// TIA Portal V17 export
// export: Created 2021-12-03T08:12:53.967625Z, ExportSetting WithDefaults, DisplayName Totally Integrated Automation Portal, DisplayVersion V17, DisplayName TIA Portal Openness, DisplayVersion V17, DisplayName TIA Portal Version Control Interface, DisplayVersion V17, DisplayName STEP 7 Professional, DisplayVersion V17, DisplayName STEP 7 Safety, DisplayVersion V17, DisplayName WinCC Advanced, DisplayVersion V17
FUNCTION "FC_DetLineCommunication_V2" : Void   // FC20, FBD
VERSION : 0.1
// stored: AutoNumber false, IsIECCheckEnabled false, UDAEnableTagReadback false
   VAR CONSTANT
      Speed_Convert : Int := 6;
   END_VAR
BEGIN

REGION Network 1: Detector Line: Start Request
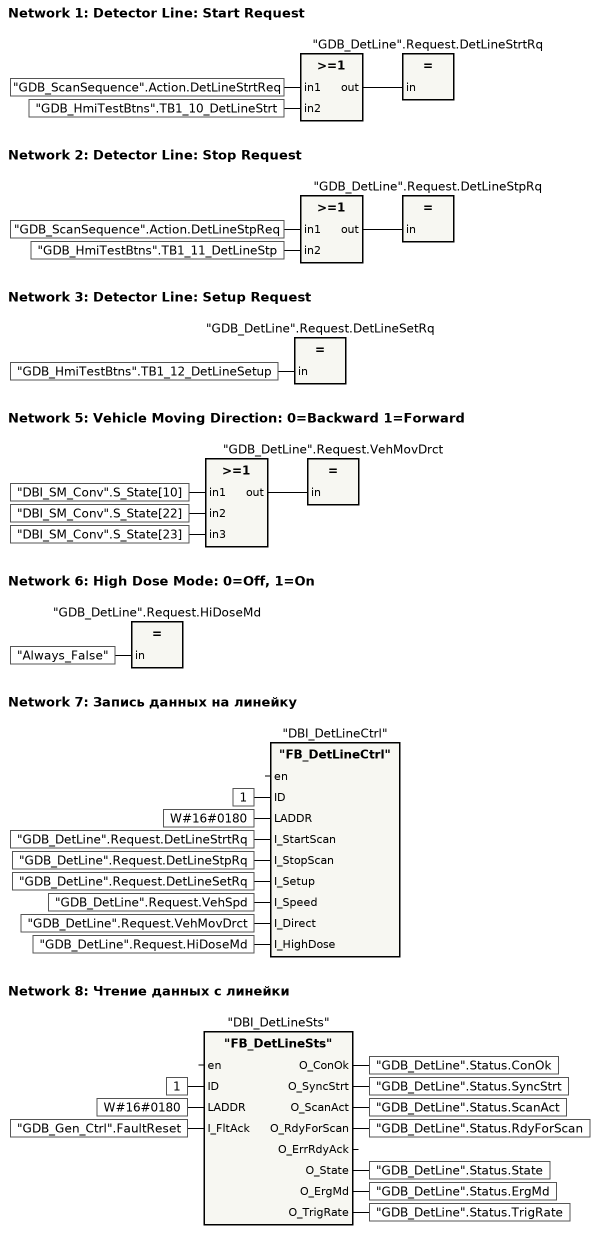
   "GDB_DetLine".Request.DetLineStrtRq := "GDB_ScanSequence".Action.DetLineStrtReq OR "GDB_HmiTestBtns".TB1_10_DetLineStrt;
END_REGION

REGION Network 2: Detector Line: Stop Request
   "GDB_DetLine".Request.DetLineStpRq := "GDB_ScanSequence".Action.DetLineStpReq OR "GDB_HmiTestBtns".TB1_11_DetLineStp;
END_REGION

REGION Network 3: Detector Line: Setup Request
   "GDB_DetLine".Request.DetLineSetRq := "GDB_HmiTestBtns".TB1_12_DetLineSetup;
END_REGION

NETWORK
TITLE = Пересчет скорости
      L     "GDB_HMI_IO_Retain".FrqConv.FastSpeed;
      L     6;
      *I;
      T     "GDB_DetLine".Request.VehSpd;

      L     "GDB_DetLine".Request.VehSpd;
      L     100;
      /I;
      T     "GDB_DetLine".Request.VehSpd;

REGION Network 5: Vehicle Moving Direction: 0=Backward 1=Forward
   "GDB_DetLine".Request.VehMovDrct := "DBI_SM_Conv".S_State[10] OR "DBI_SM_Conv".S_State[22] OR "DBI_SM_Conv".S_State[23];
END_REGION

REGION Network 6: High Dose Mode: 0=Off, 1=On
   "GDB_DetLine".Request.HiDoseMd := "Always_False";
END_REGION

REGION Network 7: Запись данных на линейку
   "DBI_DetLineCtrl"(ID := 1,   // "FB_DetLineCtrl"
                     LADDR := W#16#0180,
                     I_StartScan := "GDB_DetLine".Request.DetLineStrtRq,
                     I_StopScan := "GDB_DetLine".Request.DetLineStpRq,
                     I_Setup := "GDB_DetLine".Request.DetLineSetRq,
                     I_Speed := "GDB_DetLine".Request.VehSpd,
                     I_Direct := "GDB_DetLine".Request.VehMovDrct,
                     I_HighDose := "GDB_DetLine".Request.HiDoseMd);
END_REGION

REGION Network 8: Чтение данных с линейки
   "DBI_DetLineSts"(ID := 1,   // "FB_DetLineSts"
                    LADDR := W#16#0180,
                    I_FltAck := "GDB_Gen_Ctrl".FaultReset,
                    O_ConOk => "GDB_DetLine".Status.ConOk,
                    O_SyncStrt => "GDB_DetLine".Status.SyncStrt,
                    O_ScanAct => "GDB_DetLine".Status.ScanAct,
                    O_RdyForScan => "GDB_DetLine".Status.RdyForScan,
                    O_State => "GDB_DetLine".Status.State,
                    O_ErgMd => "GDB_DetLine".Status.ErgMd,
                    O_TrigRate => "GDB_DetLine".Status.TrigRate);
END_REGION

NETWORK
TITLE = 1=Ошибка
      L     "GDB_DetLine".Status.State;
      L     0;
      ==I;
      =     "GDB_DetLine".Status.Error;

      L     "GDB_DetLine".Status.State;
      L     1;
      ==I;
      =     "GDB_DetLine".Status.SrvsMd;

      L     "GDB_DetLine".Status.State;
      L     2;
      ==I;
      =     "GDB_DetLine".Status.AutoMd;

END_FUNCTION
